INTERFACE IEcTask EXTENDS ITask

PROPERTY NetID : amsnetid
GET
END_GET
SET
END_SET
END_PROPERTY

END_INTERFACE

(* stored: Version 1.1.0.1, ProductVersion 3.1.4024.11
   Itf IEcTask: Id {c19ff4be-e38a-4656-847e-f09011d5c178}
   Property NetID: Id {d505651c-d924-4547-8888-57722294962e}
   Get Get: Id {55b90e02-4558-45d6-bfdb-c7bec09eff38}
   Set Set: Id {28e01517-5642-4487-8593-b04cbaf78745} *)
